RoboDK station: RDTSDemoBasketLine.rdk

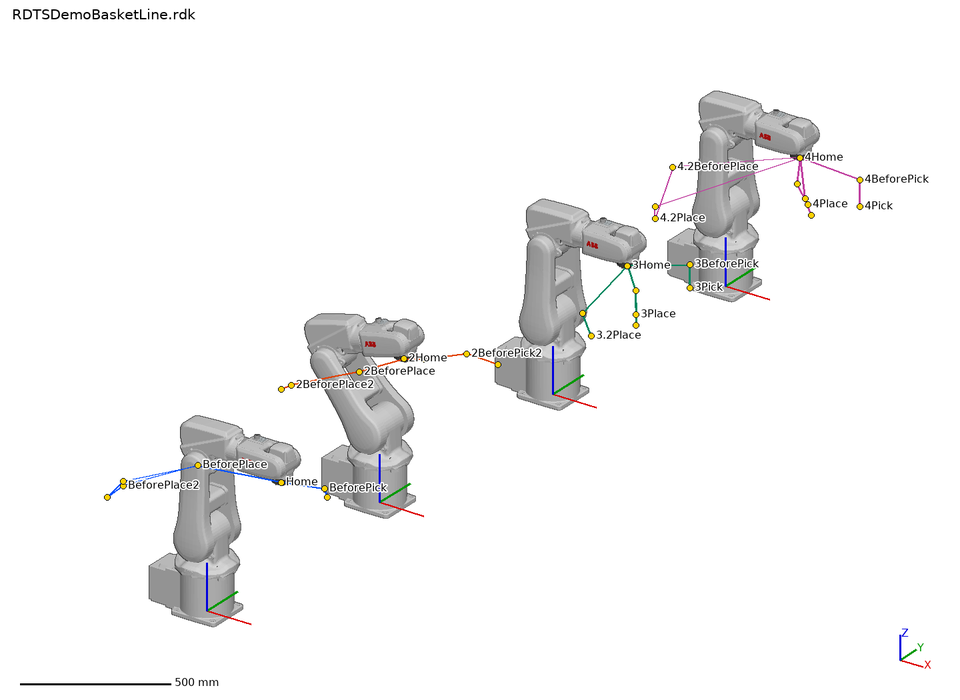
[picture v0: the station drawn from its stored meshes, robots at their saved joint values, targets as dots, program paths as lines]
Station RDTSDemoBasketLine (saved by RoboDK 5.6.7). Poses are relative to the parent item; angles as X-Y-Z fixed-axis rotations.
Station parameters (name, value as stored): 1MoveToPick, 0, 1MakePick, 0, 1PickObjOK, 1, 1MoveToPlace, 0, 1MakePlace, 0, 1PlaceObjOK, 0, 1Waitting, 1, 2MoveToPick, 0, 2MakePick, 0, 2PickObjOK, 0, 2MoveToPlace, 0, 2MakePlace, 0, 2PlaceObjOK, 0, 2Waitting, 1, 3MoveToPick, 0, 3MakePick, 0, 3PickObjOK, 0, 3MoveToPlace, 0, 3MakePlace, 0, 3PlaceObjOK, 0, 3Waitting, 1, 4MoveToPick, 0, 4MakePick, 0, 4PickObjOK, 0, 4MoveToPlace, 0, 4MakePlace, 0, 4PlaceObjOK, 0, 4Waitting, 1
  - frame Robot1Base at (0, 0, 0) mm
    - robot Robot1 (model ABB IRB 120-3/0.6): 6 axes, payload 3 kg, reach 580 mm, repeatability 0.01 mm, weight 25 kg
        modified DH rows (alpha deg, a mm, theta deg, d mm): 0, 0, 0, 290; -90, 0, -90, 0; 0, 270, 0, 0; -90, 70, 0, 302; 90, 0, 0, 0; -90, 0, 180, 72
        joint limits [-165, -110, -90, -160, -120, -400] to [165, 110, 70, 160, 120, 400]; home [0, 0, 0, 0, 0, 0]; saved at [0, 0, 0, 0, 90, 0]
    - target Home (Cartesian target) at (302, 0, 558) mm, rotated rx 180 ry 0 rz -180 deg; joints [0, 0, 0, 0, 90, 0] of Robot1
    - target BeforePick (Cartesian target) at (403.62, 104.76, 521.84) mm, rotated rx 179.56 ry -0.69 rz -179.99 deg; joints [14.447, 24.813, -22.689, 0.602, 88.437, 14.424] of Robot1
    - target Pick (Cartesian target) at (413.42, 104.99, 492) mm, rotated rx 179.56 ry -0.69 rz -179.99 deg; joints [14.149, 26.117, -18.91, 0.603, 83.358, 14.073] of Robot1
    - target AfterPick (Cartesian target) at (403.62, 104.76, 521.84) mm, rotated rx 179.56 ry -0.69 rz -179.99 deg; joints [14.447, 24.813, -22.689, 0.602, 88.437, 14.424] of Robot1
    - target BeforePlace (Cartesian target) at (0.58, -52.76, 557.96) mm, rotated rx 180 ry 0.01 rz 90.63 deg; joints [-89.37, -50.37, 30.66, 0, 109.7, 0] of Robot1
    - target BeforePlace2 (Cartesian target) at (-187.16, -214.5, 494.08) mm, rotated rx -180 ry 0.01 rz 90.63 deg; joints [-131.107, -5.367, 17.074, 0.007, 78.285, -41.739] of Robot1
    - target Place (Cartesian target) at (-181.61, -317.37, 493.69) mm, rotated rx -180 ry 0.01 rz 90.63 deg; joints [-119.781, 11.938, -1.021, 0.005, 79.074, -30.411] of Robot1
    - target AfterPlace (Cartesian target) at (-187.16, -214.5, 511.71) mm, rotated rx -180 ry 0.01 rz 90.63 deg; joints [-131.108, -5.174, 13.633, 0.007, 81.533, -41.739] of Robot1
    - target AfterPlace2 (Cartesian target) at (0.58, -52.76, 557.96) mm, rotated rx -180 ry 0.01 rz 90.63 deg; joints [-89.37, -50.37, 30.66, 0, 109.7, 0] of Robot1
  - program RobotProg1 (30 instructions, listed below)
  - frame Robot2Base at (0, 1000, 0) mm
    - robot Robot2 (model ABB IRB 120-3/0.6): 6 axes, payload 3 kg, reach 580 mm, repeatability 0.01 mm, weight 25 kg
        modified DH rows (alpha deg, a mm, theta deg, d mm): 0, 0, 0, 290; -90, 0, -90, 0; 0, 270, 0, 0; -90, 70, 0, 302; 90, 0, 0, 0; -90, 0, 180, 72
        joint limits [-165, -110, -90, -160, -120, -400] to [165, 110, 70, 160, 120, 400]; home [0, 0, 0, 0, 0, 0]; saved at [0, -40.936, 28.088, 0, 105.49, 0]
    - target 2Home (Cartesian target) at (98.64, 0, 557.45) mm, rotated rx 180 ry -2.64 rz 180 deg; joints [0, -40.936, 28.088, 0, 105.49, 0] of Robot2
    - target 2BeforePick (Cartesian target) at (141.38, 49.31, 548.14) mm, rotated rx 180 ry 0.22 rz -180 deg; joints [19.26, -32.099, 26.054, -0.072, 95.841, 19.253] of Robot2
    - target 2BeforePick2 (Cartesian target) at (172.93, 256.56, 494.82) mm, rotated rx 180 ry 0.22 rz -180 deg; joints [56.061, -0.146, 11.935, -0.184, 78.09, 56.098] of Robot2
    - target 2Pick (Cartesian target) at (298.21, 256.56, 490.23) mm, rotated rx 180 ry 0.22 rz -180 deg; joints [40.732, 18.028, -7.841, -0.144, 79.649, 40.758] of Robot2
    - target 2AfterPick (Cartesian target) at (172.93, 256.56, 494.82) mm, rotated rx 180 ry 0.22 rz -180 deg; joints [56.061, -0.146, 11.935, -0.184, 78.09, 56.098] of Robot2
    - target 2AfterPick2 (Cartesian target) at (141.38, 49.31, 548.14) mm, rotated rx 180 ry 0.22 rz -180 deg; joints [19.26, -32.099, 26.054, -0.072, 95.841, 19.253] of Robot2
    - target 2BeforePlace (Cartesian target) at (0, -119.82, 529.74) mm, rotated rx 180 ry 7.66 rz 90 deg; joints [-90, -41.74, 34.08, 0, 90, 0] of Robot2
    - target 2BeforePlace2 (Cartesian target) at (-102.6, -366.25, 550.56) mm, rotated rx -179.99 ry -0.97 rz 89.29 deg; joints [-105.6, 17.39, -18.32, -0.26, 91.86, -14.9] of Robot2
    - target 2Place (Cartesian target) at (-103.29, -422.83, 557.03) mm, rotated rx -179.99 ry -0.97 rz 89.29 deg; joints [-103.69, 33.186, -41.525, -0.232, 99.277, -13.019] of Robot2
    - target 2AfterPlace (Cartesian target) at (-102.6, -366.25, 550.56) mm, rotated rx -179.99 ry -0.97 rz 89.29 deg; joints [-105.6, 17.39, -18.32, -0.26, 91.86, -14.9] of Robot2
    - target 2AfterPlace2 (Cartesian target) at (0, -119.82, 529.74) mm, rotated rx 180 ry 7.66 rz 90 deg; joints [-90, -41.74, 34.08, 0, 90, 0] of Robot2
  - program RobotProg2 (32 instructions, listed below)
  - frame Robot3Base at (0, 2000, 0) mm
    - robot Robot3 (model ABB IRB 120-3/0.6): 6 axes, payload 3 kg, reach 580 mm, repeatability 0.01 mm, weight 25 kg
        modified DH rows (alpha deg, a mm, theta deg, d mm): 0, 0, 0, 290; -90, 0, -90, 0; 0, 270, 0, 0; -90, 70, 0, 302; 90, 0, 0, 0; -90, 0, 180, 72
        joint limits [-165, -110, -90, -160, -120, -400] to [165, 110, 70, 160, 120, 400]; home [0, 0, 0, 0, 0, 0]; saved at [0, 0, 0, 0, 90, 0]
    - target 3Home (Cartesian target) at (302, 0, 558) mm, rotated rx 180 ry 0 rz -180 deg; joints [0, 0, 0, 0, 90, 0] of Robot3
    - target 3BeforePick (Cartesian target) at (367.83, 266.67, 474.09) mm, rotated rx -179.62 ry 0.29 rz -90.13 deg; joints [35.94, 32.486, -24.68, 0.01, 81.715, -53.928] of Robot3
    - target 3Pick (Cartesian target) at (368.4, 267.1, 388.62) mm, rotated rx -179.62 ry 0.29 rz -90.13 deg; joints [35.942, 33.555, -10.401, 0.011, 66.366, -53.929] of Robot3
    - target 3AfterPick (Cartesian target) at (367.83, 266.67, 474.09) mm, rotated rx -179.62 ry 0.29 rz -90.13 deg; joints [35.94, 32.486, -24.68, 0.01, 81.715, -53.928] of Robot3
    - target 3BeforePlace (Cartesian target) at (367.85, -44.24, 503.74) mm, rotated rx -179.54 ry 0.5 rz -180 deg; joints [-6.78, 12.978, -4.113, -0.406, 80.585, -6.718] of Robot3
    - target 3Place (Cartesian target) at (368.62, -44.96, 415.73) mm, rotated rx -179.54 ry 0.5 rz -180 deg; joints [-6.876, 14.43, 10.489, -0.443, 64.531, -6.689] of Robot3
    - target 3AfterPlace (Cartesian target) at (367.85, -44.24, 503.74) mm, rotated rx -179.54 ry 0.5 rz -180 deg; joints [-6.78, 12.978, -4.113, -0.406, 80.585, -6.718] of Robot3
    - target 3.2BeforePick (Cartesian target) at (367.85, -44.24, 503.74) mm, rotated rx -179.54 ry 0.5 rz -180 deg; joints [-6.78, 12.978, -4.113, -0.406, 80.585, -6.718] of Robot3
    - target 3.2Pick (Cartesian target) at (368.97, -45.28, 375.69) mm, rotated rx -179.54 ry 0.5 rz -180 deg; joints [-6.919, 16.769, 15.263, -0.474, 57.417, -6.667] of Robot3
    - target 3.2AfterPick (Cartesian target) at (367.85, -44.24, 503.74) mm, rotated rx -179.54 ry 0.5 rz -180 deg; joints [-6.78, 12.978, -4.113, -0.406, 80.585, -6.718] of Robot3
    - target 3.2BeforePlace (Cartesian target) at (325.6, -293.23, 506.98) mm, rotated rx -179.54 ry 0.5 rz -180 deg; joints [-42.004, 29.255, -26.125, -0.01, 86.19, -42.006] of Robot3
    - target 3.2Place (Cartesian target) at (360.51, -293.82, 433.67) mm, rotated rx -179.54 ry 0.5 rz -180 deg; joints [-39.174, 34.848, -20.705, -0.045, 75.177, -39.165] of Robot3
    - target 3.2AfterPlace (Cartesian target) at (325.6, -293.23, 506.98) mm, rotated rx -179.54 ry 0.5 rz -180 deg; joints [-42.004, 29.255, -26.125, -0.01, 86.19, -42.006] of Robot3
  - program RobotProg3 (55 instructions, listed below)
  - frame Robot4Base at (0, 3000, 0) mm
    - robot Robot4 (model ABB IRB 120-3/0.6): 6 axes, payload 3 kg, reach 580 mm, repeatability 0.01 mm, weight 25 kg
        modified DH rows (alpha deg, a mm, theta deg, d mm): 0, 0, 0, 290; -90, 0, -90, 0; 0, 270, 0, 0; -90, 70, 0, 302; 90, 0, 0, 0; -90, 0, 180, 72
        joint limits [-165, -110, -90, -160, -120, -400] to [165, 110, 70, 160, 120, 400]; home [0, 0, 0, 0, 0, 0]; saved at [0, 0, 0, 0, 90, 0]
    - target 4Home (Cartesian target) at (302, 0, 558) mm, rotated rx 180 ry 0 rz -180 deg; joints [0, 0, 0, 0, 90, 0] of Robot4
    - target 4BeforePick (Cartesian target) at (382.62, 228.7, 407.15) mm, rotated rx 179.99 ry 0.01 rz -179.7 deg; joints [30.867, 30.904, -9.971, 0.001, 69.057, 30.567] of Robot4
    - target 4Pick (Cartesian target) at (382.64, 228.71, 309.5) mm, rotated rx 179.99 ry 0.01 rz -179.7 deg; joints [30.867, 36.842, -0.097, 0.001, 53.245, 30.567] of Robot4
    - target 4AfterPick (Cartesian target) at (382.62, 228.7, 407.15) mm, rotated rx 179.99 ry 0.01 rz -179.7 deg; joints [30.867, 30.904, -9.971, 0.001, 69.057, 30.567] of Robot4
    - target 4BeforePlace (Cartesian target) at (401.5, -161.2, 552.3) mm, rotated rx 180 ry 0 rz -179.65 deg; joints [-21.875, 31.361, -37.862, 0, 96.501, -22.225] of Robot4
    - target 4Place (Cartesian target) at (445.5, -160.93, 490.22) mm, rotated rx 180 ry 0 rz -179.65 deg; joints [-19.861, 39.033, -37.611, 0, 88.578, -20.211] of Robot4
    - target 4AfterPlace (Cartesian target) at (401.5, -161.2, 552.3) mm, rotated rx 180 ry 0 rz -179.65 deg; joints [-21.875, 31.361, -37.862, 0, 96.501, -22.225] of Robot4
    - target 4.2BeforePick (Cartesian target) at (433.79, -161, 508.22) mm, rotated rx 180 ry 0 rz -179.65 deg; joints [-20.363, 36.776, -37.529, 0, 90.752, -20.713] of Robot4
    - target 4.2Pick (Cartesian target) at (458.76, -160.85, 454.48) mm, rotated rx 180 ry 0 rz -179.65 deg; joints [-19.322, 41.227, -34.363, 0, 83.136, -19.672] of Robot4
    - target 4.2AfterPick (Cartesian target) at (433.79, -161, 508.22) mm, rotated rx 180 ry 0 rz -179.65 deg; joints [-20.363, 36.776, -37.529, 0, 90.752, -20.713] of Robot4
    - target 4.2BeforePlace (Cartesian target) at (-2.74, -301.99, 558) mm, rotated rx 180 ry 0 rz 89.48 deg; joints [-90.52, 0, 0, 0, 90, 0] of Robot4
    - target 4.2Place (Cartesian target) at (-3.66, -402.77, 408.42) mm, rotated rx 180 ry 0 rz 89.48 deg; joints [-90.52, 21.468, 2.901, 0, 65.631, 0] of Robot4
    - target 4.2AfterPlace (Cartesian target) at (-3.66, -402.77, 453.53) mm, rotated rx 180 ry 0 rz 89.48 deg; joints [-90.52, 20.215, -3.866, 0, 73.651, 0] of Robot4
  - program RobotProg4 (55 instructions, listed below)
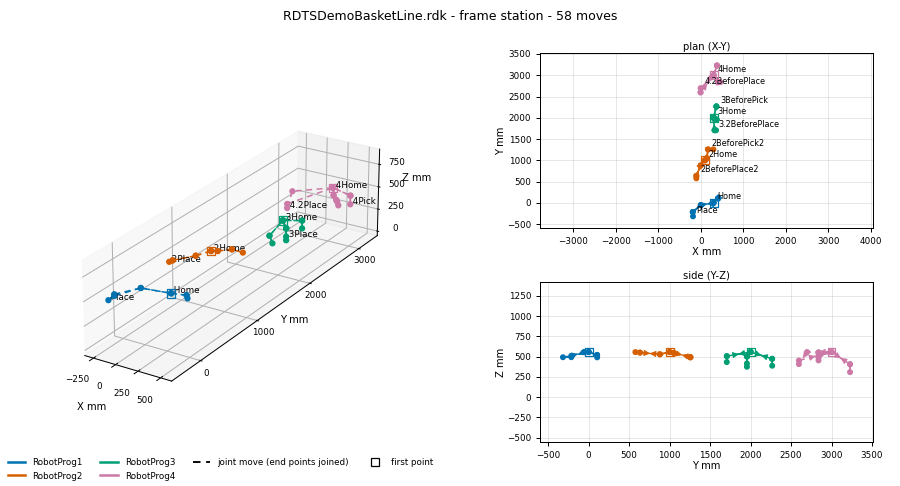
[picture p0: tool path of RDTSDemoBasketLine.rdk in frame station, 58 of 58 moves have a stored position in this frame; points joined in program order, loops and branches not executed]

--- program RobotProg1 (robot Robot1) ---
  设置参考: Robot1Base
  MoveJ (Home)
  Set 1MakePick=0
  Set 1PickObjOK=0
  Set 1MakePlace=0
  Set 1PlaceObjOK=0
  Wait 1MoveToPick=1
  Set 1Waitting=0
  MoveJ (BeforePick)
  MoveJ (Pick)
  Set 1MakePick=1
  Wait 1PickObjOK=1
  Set 1MakePick=0
  暂停 2.0 s
  MoveJ (AfterPick)
  MoveJ (Home)
  Set 1Waitting=1
  Wait 1MoveToPlace=1
  Set 1Waitting=0
  MoveJ (BeforePlace)
  MoveJ (BeforePlace2)
  MoveJ (Place)
  Set 1MakePlace=1
  Wait 1PlaceObjOK=1
  Set 1MakePlace=0
  暂停 1.0 s
  MoveJ (AfterPlace)
  MoveJ (AfterPlace2)
  MoveJ (Home)
  Set 1Waitting=1

--- program RobotProg2 (robot Robot2) ---
  设置参考: Robot2Base
  MoveJ (2Home)
  Set 2MakePick=0
  Set 2PickObjOK=0
  Set 2MakePlace=0
  Set 2PlaceObjOK=0
  Wait 2MoveToPick=1
  Set 2Waitting=0
  MoveJ (2BeforePick)
  MoveJ (2BeforePick2)
  MoveJ (2Pick)
  Set 2MakePick=1
  Wait 2PickObjOK=1
  Set 2MakePick=0
  暂停 2.0 s
  MoveJ (2AfterPick)
  MoveJ (2AfterPick2)
  MoveJ (2Home)
  Set 2Waitting=1
  Wait 2MoveToPlace=1
  Set 2Waitting=0
  MoveJ (2BeforePlace)
  MoveJ (2BeforePlace2)
  MoveJ (2Place)
  Set 2MakePlace=1
  Wait 2PlaceObjOK=1
  Set 2MakePlace=0
  暂停 1.0 s
  MoveJ (2AfterPlace)
  MoveJ (2AfterPlace2)
  MoveJ (2Home)
  Set 2Waitting=1

--- program RobotProg3 (robot Robot3) ---
  设置参考: Robot3Base
  MoveJ (3Home)
  Set 3MakePick=0
  Set 3PickObjOK=0
  Set 3MakePlace=0
  Set 3PlaceObjOK=0
  Wait 3MoveToPick=1
  Set 3Waitting=0
  MoveJ (3BeforePick)
  MoveJ (3Pick)
  Set 3MakePick=1
  Wait 3PickObjOK=1
  Set 3MakePick=0
  暂停 2.0 s
  MoveJ (3AfterPick)
  MoveJ (3Home)
  Set 3Waitting=1
  Wait 3MoveToPlace=1
  Set 3Waitting=0
  MoveJ (3BeforePlace)
  MoveJ (3Place)
  Set 3MakePlace=1
  Wait 3PlaceObjOK=1
  Set 3MakePlace=0
  暂停 1.0 s
  MoveJ (3AfterPlace)
  MoveJ (3Home)
  Set 3Waitting=1
  暂停 2.5 s
  Set 3MakePick=0
  Set 3PickObjOK=0
  Set 3MakePlace=0
  Set 3PlaceObjOK=0
  Wait 3MoveToPick=1
  Set 3Waitting=0
  MoveJ (3.2BeforePick)
  MoveJ (3.2Pick)
  Set 3MakePick=1
  Wait 3PickObjOK=1
  Set 3MakePick=0
  暂停 2.0 s
  MoveJ (3.2AfterPick)
  MoveJ (3Home)
  Set 3Waitting=1
  Wait 3MoveToPlace=1
  Set 3Waitting=0
  MoveJ (3.2BeforePlace)
  MoveJ (3.2Place)
  Set 3MakePlace=1
  Wait 3PlaceObjOK=1
  Set 3MakePlace=0
  暂停 1.0 s
  MoveJ (3.2AfterPlace)
  MoveJ (3Home)
  Set 3Waitting=1

--- program RobotProg4 (robot Robot4) ---
  设置参考: Robot4Base
  MoveJ (4Home)
  Set 4MakePick=0
  Set 4PickObjOK=0
  Set 4MakePlace=0
  Set 4PlaceObjOK=0
  Wait 4MoveToPick=1
  Set 4Waitting=0
  MoveJ (4BeforePick)
  MoveJ (4Pick)
  Set 4MakePick=1
  Wait 4PickObjOK=1
  Set 4MakePick=0
  暂停 2.0 s
  MoveJ (4AfterPick)
  MoveJ (4Home)
  Set 4Waitting=1
  Wait 4MoveToPlace=1
  Set 4Waitting=0
  MoveJ (4BeforePlace)
  MoveJ (4Place)
  Set 4MakePlace=1
  Wait 4PlaceObjOK=1
  Set 4MakePlace=0
  暂停 1.0 s
  MoveJ (4AfterPlace)
  MoveJ (4Home)
  Set 4Waitting=1
  暂停 2.5 s
  Set 4MakePick=0
  Set 4PickObjOK=0
  Set 4MakePlace=0
  Set 4PlaceObjOK=0
  Wait 4MoveToPick=1
  Set 4Waitting=0
  MoveJ (4.2BeforePick)
  MoveJ (4.2Pick)
  Set 4MakePick=1
  Wait 4PickObjOK=1
  Set 4MakePick=0
  暂停 2.0 s
  MoveJ (4.2AfterPick)
  MoveJ (4Home)
  Set 4Waitting=1
  Wait 4MoveToPlace=1
  Set 4Waitting=0
  MoveJ (4.2BeforePlace)
  MoveJ (4.2Place)
  Set 4MakePlace=1
  Wait 4PlaceObjOK=1
  Set 4MakePlace=0
  暂停 1.0 s
  MoveJ (4.2AfterPlace)
  MoveJ (4Home)
  Set 4Waitting=1
